// TIA Portal V20 export
DATA_BLOCK "SqlData"   // DB5
TITLE = SqlData
{ S7_Optimized_Access := 'TRUE' }
AUTHOR : SIEMENS SUP Applications
VERSION : 3.0
// DB for holding the strucutured data received from a Tabular Data Stream SELECT response
// stored: MemoryReserve 0
   VAR
      data { ExternalAccessible := 'False'; ExternalVisible := 'False'; ExternalWritable := 'False'} : "typeSqlData";
   END_VAR
BEGIN
END_DATA_BLOCK
